// TIA Portal V17 export
// export: Created 2022-02-03T14:45:12.663588Z, ExportSetting WithDefaults, DisplayName Totally Integrated Automation Portal, DisplayVersion V17, DisplayName TIA Portal Openness, DisplayVersion V17, DisplayName TIA Portal Version Control Interface, DisplayVersion V17, DisplayName SINAMICS Startdrive Advanced, DisplayVersion V17, DisplayName SINAMICS Startdrive G130, G150, S120, S150, SINAMICS MV, S210, DisplayVersion V17, DisplayName SINAMICS Startdrive G110M, G120, G120C, G120D, G120P, G115D, DisplayVersion V17, DisplayName STEP 7 Professional, DisplayVersion V17, DisplayName STEP 7 Safety, DisplayVersion V17, DisplayName WinCC Advanced, DisplayVersion V17
FUNCTION_BLOCK "Statistic"   // FB5, LAD
VERSION : 0.1
// stored: Access Published, AutoNumber true, IsIECCheckEnabled false, IsRetainMemResEnabled false, MemoryReserve 100, SetENOAutomatically false, UDAEnableTagReadback false
   VAR_INPUT
      Operation : Bool;
      occupiedBay : Array["FIRSTBAY".."LASTBAY"] of Bool;
   END_VAR
   VAR_IN_OUT
      statistics : "typeStatistics";
   END_VAR
   VAR
      statOldOperation : Bool;
   END_VAR
   VAR RETAIN
      InstIEC_Counter1 { S7_SetPoint := 'True'} : CTU_UINT;
      InstIEC_Counter2 { S7_SetPoint := 'True'} : CTU_UINT;
      INSTIEC_Counter3 { S7_SetPoint := 'True'} : CTU_UINT;
   END_VAR
   VAR_TEMP
      tempRisOperation : Bool;
   END_VAR
   VAR_TEMP   // added for the SCL form of the ladder/FBD networks
      _w1 : Bool;
   END_VAR
BEGIN

REGION Network 1
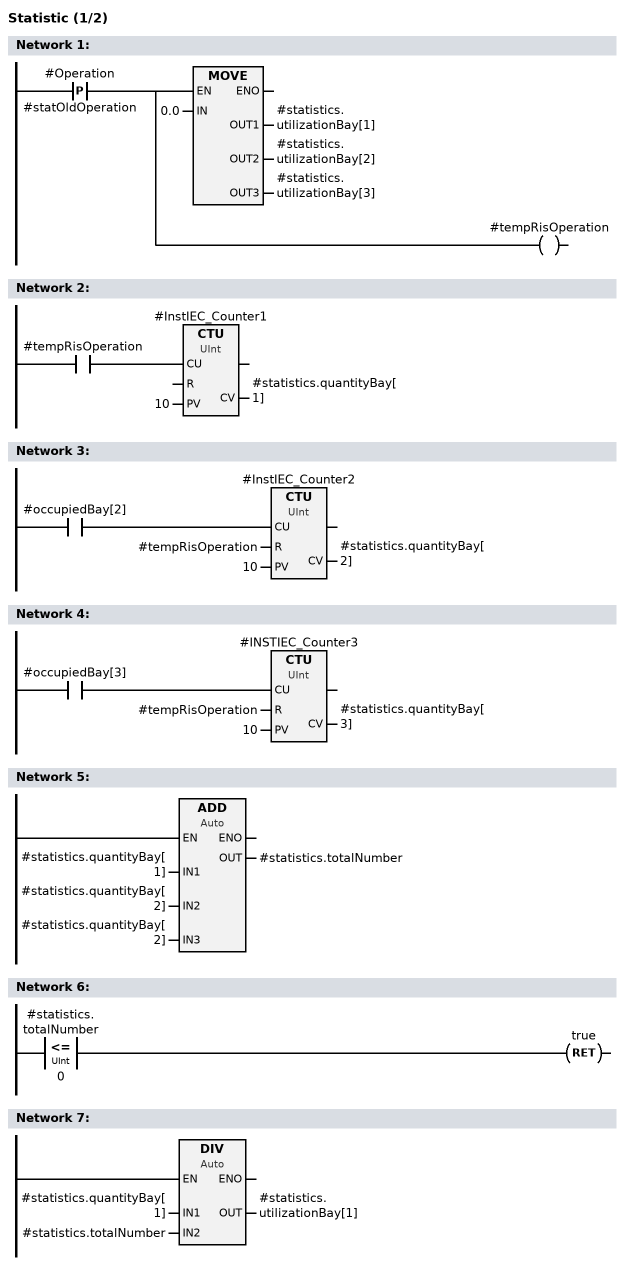
   RUNG wire#powerrail
      P_Contact(operand := #Operation, bit := #statOldOperation)
      wire#w1
      Move(in := 0.0, out1 => #statistics.utilizationBay[1], out2 => #statistics.utilizationBay[2], out3 => #statistics.utilizationBay[3])
   END_RUNG
   RUNG wire#w1
      Coil( #tempRisOperation )
   END_RUNG
   // the same network as SCL:
   #_w1 := #Operation AND NOT #statOldOperation;   // rising edge of #Operation
   #statOldOperation := #Operation;
   IF #_w1 THEN
       #statistics.utilizationBay[1] := 0.0;
       #statistics.utilizationBay[2] := 0.0;
       #statistics.utilizationBay[3] := 0.0;
   END_IF;
   #tempRisOperation := #_w1;
END_REGION

REGION Network 2
   RUNG wire#powerrail
      Contact( #tempRisOperation )
      { S7_Templates := "value_type := UInt" } #InstIEC_Counter1.CTU(r :=, pv := 10, cv => #statistics.quantityBay[1])
   END_RUNG
   // the same network as SCL:
   #InstIEC_Counter1(CU := #tempRisOperation, PV := 10, CV => #statistics.quantityBay[1]);   // CTU
END_REGION

REGION Network 3
   RUNG wire#powerrail
      Contact( #occupiedBay[2] )
      { S7_Templates := "value_type := UInt" } #InstIEC_Counter2.CTU(r := #tempRisOperation, pv := 10, cv => #statistics.quantityBay[2])
   END_RUNG
   // the same network as SCL:
   #InstIEC_Counter2(CU := #occupiedBay[2], R := #tempRisOperation, PV := 10, CV => #statistics.quantityBay[2]);   // CTU
END_REGION

REGION Network 4
   RUNG wire#powerrail
      Contact( #occupiedBay[3] )
      { S7_Templates := "value_type := UInt" } #INSTIEC_Counter3.CTU(r := #tempRisOperation, pv := 10, cv => #statistics.quantityBay[3])
   END_RUNG
   // the same network as SCL:
   #INSTIEC_Counter3(CU := #occupiedBay[3], R := #tempRisOperation, PV := 10, CV => #statistics.quantityBay[3]);   // CTU
END_REGION

REGION Network 5
   RUNG wire#powerrail
      Add(in1 := #statistics.quantityBay[1], in2 := #statistics.quantityBay[2], in3 := #statistics.quantityBay[2], out => #statistics.totalNumber)
   END_RUNG
   // the same network as SCL:
   #statistics.totalNumber := #statistics.quantityBay[1] + #statistics.quantityBay[2] + #statistics.quantityBay[2];
END_REGION

REGION Network 6
   IF #statistics.totalNumber <= 0 THEN
       ENO := true;
       RETURN;
   END_IF;
END_REGION

REGION Network 7
   RUNG wire#powerrail
      Div(in1 := #statistics.quantityBay[1], in2 := #statistics.totalNumber, out => #statistics.utilizationBay[1])
   END_RUNG
   // the same network as SCL:
   #statistics.utilizationBay[1] := #statistics.quantityBay[1] / #statistics.totalNumber;
END_REGION

REGION Network 8
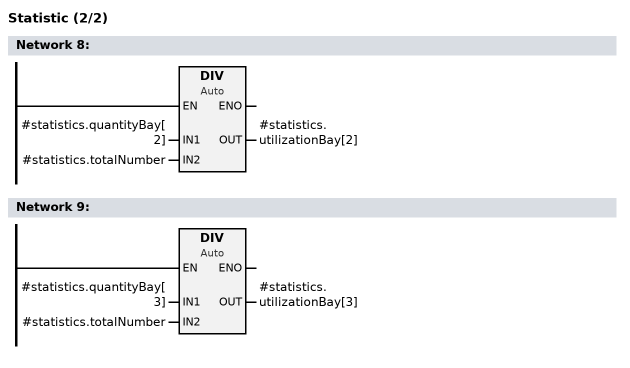
   RUNG wire#powerrail
      Div(in1 := #statistics.quantityBay[2], in2 := #statistics.totalNumber, out => #statistics.utilizationBay[2])
   END_RUNG
   // the same network as SCL:
   #statistics.utilizationBay[2] := #statistics.quantityBay[2] / #statistics.totalNumber;
END_REGION

REGION Network 9
   RUNG wire#powerrail
      Div(in1 := #statistics.quantityBay[3], in2 := #statistics.totalNumber, out => #statistics.utilizationBay[3])
   END_RUNG
   // the same network as SCL:
   #statistics.utilizationBay[3] := #statistics.quantityBay[3] / #statistics.totalNumber;
END_REGION
END_FUNCTION_BLOCK
